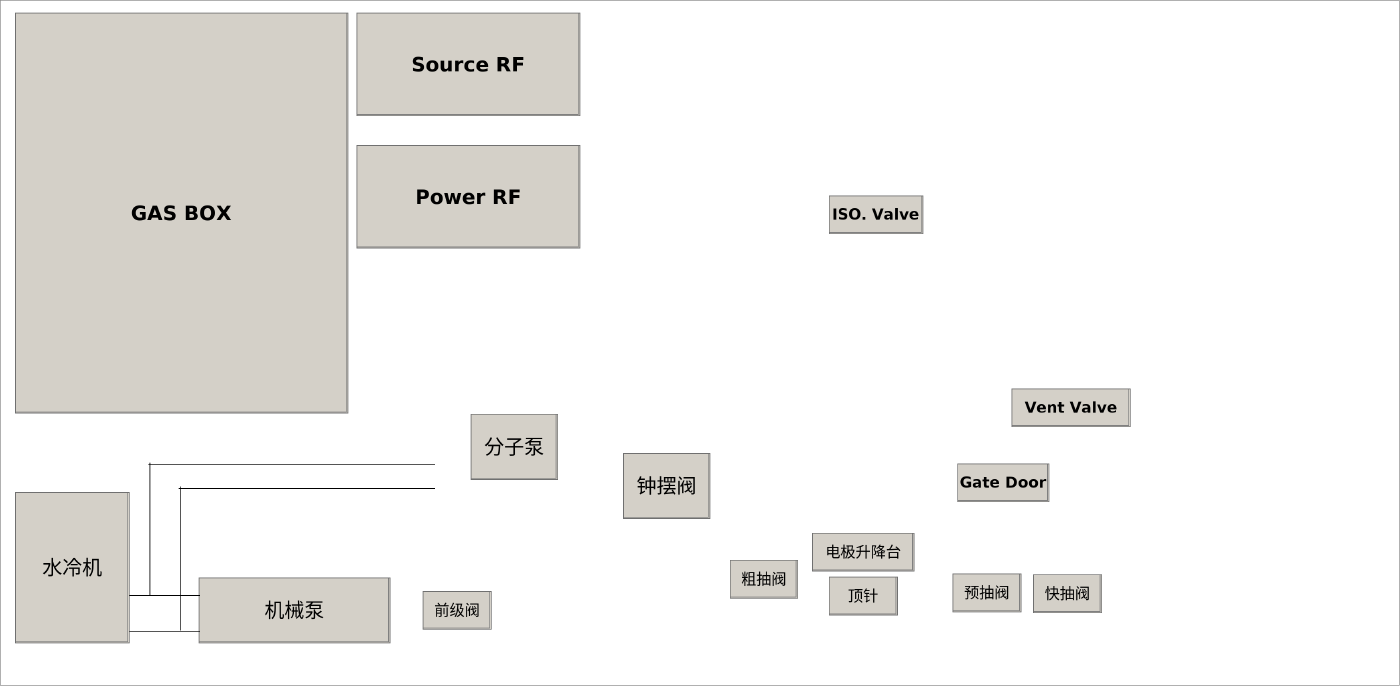
VISUALIZATION Overview_Total  // 1755x860, background image ImagePool1.autoImg
    Button (249,724 240x82), "机械泵"
    Button (19,617 143x189), "水冷机"
    Line (162,791) (250,791)
    Line (162,746) (250,746)
    Line (188,746) (188,580)
    Line (226,790) (226,610)
    Line (186,582) (545,582)
    Line (224,612) (545,612)
    Button (590,519 109x82), "分子泵"
    Button (781,568 109x82), "钟摆阀"
    Button (530,741 86x48), "前级阀"
    Button (915,702 85x48), "粗抽阀"
    Button (1018,668 128x48), "电极升降台"
    Button (1039,723 86x48), "顶针"
    Button (1194,719 86x48), "预抽阀"
    Button (1295,720 86x48), "快抽阀"
    Button (19,16 417x502), "GAS BOX"
    Button (1039,245 118x48), "ISO. Valve"
    Button (1200,581 115x48), "Gate Door"
    Button (1268,487 149x48), "Vent Valve"
    Button (447,16 280x129), "Source RF"
    Button (447,182 280x129), "Power RF"
END_VISUALIZATION

(* stored: Version 1.1.0.1, ProductVersion 3.1.4024.4
   Visu Overview_Total: Id {8c4833bf-01f9-439b-8f8e-1acb88a7cd80} *)
